(* IEC 61131-3 sources: github/IM_SYS_PRG/Code/顶出系统/托模, 2 files *)

(* ---- FB_Eject.st ---- *)
(*
  FB_Eject 功能块
  功能：
  1. 负责托模进、托模保持、托模退及其调试动作的执行状态机。
  2. 按托模参数输出压力、速度、位置命令，并返回托模进退完成状态。

  说明：
  1. 正常模式使用 1=托模进、2=托模退；调试模式使用 6/7。
  2. 组合托模模式由 `FB_EjectMode` 复用本块完成具体动作。
*)
FUNCTION_BLOCK FB_Eject
VAR_IN_OUT
    stEjectAxis: ST_AxisRefHyd;       // 托模共享轴结构
END_VAR
VAR_INPUT
    bStart: BOOL;                     // TRUE=启动托模动作
    bStop: BOOL;                      // TRUE=正常停止
    bEStop: BOOL;                     // TRUE=急停
    bReset: BOOL;                     // TRUE=复位状态机与输出
    bManualMode: BOOL;                // TRUE=手动点动托模
    uiEjectMode: UINT;                // 1=托模进 2=托模退 6=托模进调试 7=托模退调试
    stEjectPara: ST_EjectPara;        // 托模工艺参数
    bEjectInStop: BOOL;               // 托模进停止信号
    bEjectOutStop: BOOL;              // 托模退停止信号
    udiEjectElecRulerVal: UDINT;      // 位置反馈
END_VAR
VAR_OUTPUT
    bBusy: BOOL;                      // TRUE=当前动作尚未结束
    bDone: BOOL;                      // TRUE=当前动作完成
    bAlarm: BOOL;                     // TRUE=当前动作报警
    dwAlarmID: DWORD;                 // 模块报警码
    uiActHint: UINT;                  // 当前动作提示码
    uiActTime: UINT;                  // 当前动作持续时间，单位 s
    bEjectIned: BOOL;                 // TRUE=托模进完成
    bEjectOuted: BOOL;                // TRUE=托模退完成
    uiPresCmd: UINT;                  // 压力命令输出
    uiSpdCmd: UINT;                   // 速度命令输出
    udiPosCmd: UDINT;                 // 位置命令输出
END_VAR
VAR
    eState: E_EjectState := eState_Idle;
    uiStageIndex: UINT := 0;
    tPulse: TON;
    udiElapsedMs: UDINT := 0;
    bManualActive: BOOL := FALSE;
    bInRequest: BOOL := FALSE;
    bOutRequest: BOOL := FALSE;
    stSegCmd: ST_EjectSeg;
END_VAR

bManualActive := bManualMode OR (uiEjectMode = 6) OR (uiEjectMode = 7);
bInRequest := (uiEjectMode = 1) OR (uiEjectMode = 6);
bOutRequest := (uiEjectMode = 2) OR (uiEjectMode = 7);

IF bReset THEN
    eState := eState_Idle;
    bBusy := FALSE;
    bDone := FALSE;
    bAlarm := FALSE;
    dwAlarmID := 0;
    uiActHint := 0;
    uiActTime := 0;
    bEjectIned := FALSE;
    bEjectOuted := FALSE;
    uiPresCmd := 0;
    uiSpdCmd := 0;
    udiPosCmd := 0;
    uiStageIndex := 0;
    udiElapsedMs := 0;
    tPulse(IN := FALSE, PT := T#100MS);
ELSIF bEStop THEN
    eState := eState_Error;
    bAlarm := TRUE;
    dwAlarmID := dwAlarmID OR DWORD#16#0010;
    uiActHint := 1;
    uiPresCmd := 0;
    uiSpdCmd := 0;
    udiPosCmd := 0;
    tPulse(IN := FALSE, PT := T#100MS);
ELSIF bStop THEN
    eState := eState_Idle;
    bBusy := FALSE;
    uiPresCmd := 0;
    uiSpdCmd := 0;
    udiPosCmd := 0;
    uiActHint := 0;
    udiElapsedMs := 0;
    tPulse(IN := FALSE, PT := T#100MS);
ELSE
    CASE eState OF
        eState_Idle:
            bBusy := FALSE;
            bDone := FALSE;
            uiActHint := 0;
            uiActTime := 0;
            bEjectIned := FALSE;
            bEjectOuted := FALSE;
            uiPresCmd := 0;
            uiSpdCmd := 0;
            udiPosCmd := 0;
            uiStageIndex := 0;
            udiElapsedMs := 0;
            tPulse(IN := FALSE, PT := T#100MS);
            IF bStart THEN
                bAlarm := FALSE;
                dwAlarmID := 0;
                uiStageIndex := 1;
                IF bInRequest THEN
                    eState := eState_EjectIning;
                ELSIF bOutRequest THEN
                    eState := eState_EjectOuting;
                ELSE
                    bAlarm := TRUE;
                    dwAlarmID := DWORD#16#0001;
                    eState := eState_Error;
                END_IF;
            END_IF;

        eState_EjectIning:
            bBusy := TRUE;
            tPulse(IN := TRUE, PT := T#100MS);
            IF tPulse.Q THEN
                udiElapsedMs := udiElapsedMs + 100;
                tPulse(IN := FALSE, PT := T#100MS);
            END_IF;
            uiActTime := TO_UINT(udiElapsedMs / 1000);

            IF bManualActive THEN
                stSegCmd := stEjectPara.stEjectInDbgSeg;
                IF (stSegCmd.uiPres = 0) AND (stSegCmd.uiSpd = 0) AND (stSegCmd.udiPos = 0) THEN
                    stSegCmd := stEjectPara.aEjectInSeg[1];
                END_IF;
                uiActHint := 28;
                uiPresCmd := stSegCmd.uiPres;
                uiSpdCmd := stSegCmd.uiSpd;
                udiPosCmd := stSegCmd.udiPos;
                IF NOT bStart THEN
                    eState := eState_Idle;
                END_IF;
            ELSE
                IF uiStageIndex > stEjectPara.uiEjectInSegCnt THEN
                    IF stEjectPara.stEjectKeepSeg.uiTime > 0 THEN
                        eState := eState_EjectKeeping;
                    ELSE
                        eState := eState_EjectIned;
                    END_IF;
                    udiElapsedMs := 0;
                    tPulse(IN := FALSE, PT := T#100MS);
                ELSE
                    stSegCmd := stEjectPara.aEjectInSeg[uiStageIndex];
                    uiActHint := 89 + uiStageIndex; // 90-92
                    uiPresCmd := stSegCmd.uiPres;
                    uiSpdCmd := stSegCmd.uiSpd;
                    udiPosCmd := stSegCmd.udiPos;

                    IF (stEjectPara.uiEjectInMode = 2) AND (udiEjectElecRulerVal >= stSegCmd.udiPos) THEN
                        uiStageIndex := uiStageIndex + 1;
                        udiElapsedMs := 0;
                        tPulse(IN := FALSE, PT := T#100MS);
                    ELSIF ((stEjectPara.uiEjectInMode = 0) AND (stSegCmd.uiTime > 0) AND (udiElapsedMs >= TO_UDINT(stSegCmd.uiTime))) OR ((stEjectPara.uiEjectInMode = 1) AND bEjectInStop) THEN
                        uiStageIndex := uiStageIndex + 1;
                        udiElapsedMs := 0;
                        tPulse(IN := FALSE, PT := T#100MS);
                    END_IF;

                    IF (stEjectPara.uiEjectInLimitTime > 0) AND (udiElapsedMs >= TO_UDINT(stEjectPara.uiEjectInLimitTime)) THEN
                        dwAlarmID := dwAlarmID OR DWORD#16#0001;
                        eState := eState_Error;
                    END_IF;
                END_IF;
            END_IF;

        eState_EjectIned:
            bBusy := FALSE;
            bDone := TRUE;
            bEjectIned := TRUE;
            uiActHint := 30;
            uiPresCmd := 0;
            uiSpdCmd := 0;
            udiPosCmd := 0;

        eState_EjectKeeping:
            bBusy := TRUE;
            uiActHint := 29;
            uiPresCmd := stEjectPara.stEjectKeepSeg.uiPres;
            uiSpdCmd := stEjectPara.stEjectKeepSeg.uiSpd;
            udiPosCmd := stEjectPara.stEjectKeepSeg.udiPos;
            tPulse(IN := TRUE, PT := T#100MS);
            IF tPulse.Q THEN
                udiElapsedMs := udiElapsedMs + 100;
                tPulse(IN := FALSE, PT := T#100MS);
            END_IF;
            uiActTime := TO_UINT(udiElapsedMs / 1000);
            IF (stEjectPara.stEjectKeepSeg.uiTime = 0) OR (udiElapsedMs >= TO_UDINT(stEjectPara.stEjectKeepSeg.uiTime)) THEN
                eState := eState_EjectKept;
                tPulse(IN := FALSE, PT := T#100MS);
            END_IF;

        eState_EjectKept:
            bBusy := FALSE;
            bDone := TRUE;
            bEjectIned := TRUE;
            uiActHint := 29;
            uiPresCmd := 0;
            uiSpdCmd := 0;
            udiPosCmd := 0;

        eState_EjectOuting:
            bBusy := TRUE;
            tPulse(IN := TRUE, PT := T#100MS);
            IF tPulse.Q THEN
                udiElapsedMs := udiElapsedMs + 100;
                tPulse(IN := FALSE, PT := T#100MS);
            END_IF;
            uiActTime := TO_UINT(udiElapsedMs / 1000);

            IF bManualActive THEN
                stSegCmd := stEjectPara.stEjectOutDbgSeg;
                IF (stSegCmd.uiPres = 0) AND (stSegCmd.uiSpd = 0) AND (stSegCmd.udiPos = 0) THEN
                    stSegCmd := stEjectPara.aEjectOutSeg[1];
                END_IF;
                uiActHint := 31;
                uiPresCmd := stSegCmd.uiPres;
                uiSpdCmd := stSegCmd.uiSpd;
                udiPosCmd := stSegCmd.udiPos;
                IF NOT bStart THEN
                    eState := eState_Idle;
                END_IF;
            ELSE
                IF uiStageIndex > stEjectPara.uiEjectOutSegCnt THEN
                    eState := eState_EjectOuted;
                ELSE
                    stSegCmd := stEjectPara.aEjectOutSeg[uiStageIndex];
                    uiActHint := 91 + uiStageIndex; // 92-94
                    uiPresCmd := stSegCmd.uiPres;
                    uiSpdCmd := stSegCmd.uiSpd;
                    udiPosCmd := stSegCmd.udiPos;

                    IF (stEjectPara.uiEjectOutMode = 2) AND (udiEjectElecRulerVal >= stSegCmd.udiPos) THEN
                        uiStageIndex := uiStageIndex + 1;
                        udiElapsedMs := 0;
                        tPulse(IN := FALSE, PT := T#100MS);
                    ELSIF ((stEjectPara.uiEjectOutMode = 0) AND (stSegCmd.uiTime > 0) AND (udiElapsedMs >= TO_UDINT(stSegCmd.uiTime))) OR ((stEjectPara.uiEjectOutMode = 1) AND bEjectOutStop) THEN
                        uiStageIndex := uiStageIndex + 1;
                        udiElapsedMs := 0;
                        tPulse(IN := FALSE, PT := T#100MS);
                    END_IF;

                    IF (stEjectPara.uiEjectOutLimitTime > 0) AND (udiElapsedMs >= TO_UDINT(stEjectPara.uiEjectOutLimitTime)) THEN
                        dwAlarmID := dwAlarmID OR DWORD#16#0002;
                        eState := eState_Error;
                    END_IF;
                END_IF;
            END_IF;

        eState_EjectOuted:
            bBusy := FALSE;
            bDone := TRUE;
            bEjectOuted := TRUE;
            uiActHint := 32;
            uiPresCmd := 0;
            uiSpdCmd := 0;
            udiPosCmd := 0;

        eState_Error:
            bBusy := FALSE;
            bAlarm := TRUE;
            uiActHint := 1;
            uiPresCmd := 0;
            uiSpdCmd := 0;
            udiPosCmd := 0;
            tPulse(IN := FALSE, PT := T#100MS);

    ELSE
        eState := eState_Error;
    END_CASE;
END_IF;

stEjectAxis.rSetPressure := TO_LREAL(uiPresCmd);
stEjectAxis.rSetVelocity := TO_LREAL(uiSpdCmd);
stEjectAxis.rSetPosition := TO_LREAL(udiPosCmd);
stEjectAxis.stPumpRequest.bRequest := bBusy;
stEjectAxis.stPumpRequest.rPressureSet := TO_LREAL(uiPresCmd);
stEjectAxis.stPumpRequest.rFlowSet := TO_LREAL(uiSpdCmd);
IF bBusy THEN
    stEjectAxis.eAxisState := Running;
ELSE
    stEjectAxis.eAxisState := Idle;
END_IF;
stEjectAxis.nFaultCode := TO_INT(dwAlarmID);
END_FUNCTION_BLOCK

(* ---- FB_EjectMode.st ---- *)
(*
  FB_EjectMode 功能块
  功能：
  1. 在基础 `FB_Eject` 之上组合出定次、震动、停留三种托模模式。
  2. 通过内部顺序控制，把“托模进/托模退/托模保持”拼成更高层动作。
  3. 对外仍保持与普通托模模块相似的 Busy/Done/Alarm 接口，便于主控统一调用。

  说明：
  1. 本块本身不直接生成液压命令，而是复用 `FB_Eject` 完成具体动作。
  2. `uiSeqPhase` 用来表示当前执行到“复位子块、托进、再次复位、托退”的哪一步。
  3. 只有在手动组合模式被上层明确选择时，才应该让本块接管托模轴输出。
*)
FUNCTION_BLOCK FB_EjectMode
VAR_IN_OUT
    stEjectAxis: ST_AxisRefHyd;
END_VAR
VAR_INPUT
    bStart: BOOL;
    bStop: BOOL;
    bEStop: BOOL;
    bReset: BOOL;
    uiEjectMode: UINT;            // 1=定次 2=震动 3=停留
    uiEjectTimes: UINT;           // 定次/震动次数；震动模式下 0 表示持续循环
    stEjectPara: ST_EjectPara;
    bEjectInStop: BOOL;
    bEjectOutStop: BOOL;
    udiEjectElecRulerVal: UDINT;
END_VAR
VAR_OUTPUT
    bBusy: BOOL;
    bDone: BOOL;
    bAlarm: BOOL;
    dwAlarmID: DWORD;
    uiActHint: UINT;
    uiActTime: UINT;
    bEjectIned: BOOL;
    bEjectOuted: BOOL;
    uiPresCmd: UINT;
    uiSpdCmd: UINT;
    udiPosCmd: UDINT;
END_VAR
VAR
    eState: E_EjectModeState := eState_Idle;
    fbEject: FB_Eject;

    (* 发给内部 `FB_Eject` 的命令。 *)
    bCmdStart: BOOL := FALSE;
    bCmdReset: BOOL := FALSE;
    uiCmdMode: UINT := 0;

    (* 顺序控制变量。 *)
    uiExecCount: UINT := 0;
    uiSeqPhase: UINT := 0;

    (* 内部 `FB_Eject` 状态缓存。 *)
    bSubBusy: BOOL := FALSE;
    bSubDone: BOOL := FALSE;
    bSubAlarm: BOOL := FALSE;
    dwSubAlarmID: DWORD := 0;
    uiSubActHint: UINT := 0;
    uiSubActTime: UINT := 0;
    bSubEjectIned: BOOL := FALSE;
    bSubEjectOuted: BOOL := FALSE;
    uiSubPresCmd: UINT := 0;
    uiSubSpdCmd: UINT := 0;
    udiSubPosCmd: UDINT := 0;
END_VAR

(* 每个扫描周期先清空对子块的控制命令。 *)
bCmdStart := FALSE;
bCmdReset := FALSE;
uiCmdMode := 0;

IF bReset THEN
    eState := eState_Idle;
    bBusy := FALSE;
    bDone := FALSE;
    bAlarm := FALSE;
    dwAlarmID := DWORD#0;
    uiActHint := 0;
    uiActTime := 0;
    uiExecCount := 0;
    uiSeqPhase := 0;
    bCmdReset := TRUE;

ELSIF bEStop THEN
    eState := eState_Error;
    bBusy := FALSE;
    bDone := FALSE;
    bAlarm := TRUE;
    dwAlarmID := DWORD#16#0010;
    uiActHint := 1;
    uiActTime := 0;
    uiExecCount := 0;
    uiSeqPhase := 0;
    bCmdReset := TRUE;

ELSIF bStop THEN
    eState := eState_Idle;
    bBusy := FALSE;
    bDone := FALSE;
    bAlarm := FALSE;
    dwAlarmID := DWORD#0;
    uiActHint := 0;
    uiActTime := 0;
    uiExecCount := 0;
    uiSeqPhase := 0;
    bCmdReset := TRUE;

ELSE
    CASE eState OF
        eState_Idle:
            bBusy := FALSE;
            uiActHint := 0;
            uiActTime := 0;

            IF bStart THEN
                bDone := FALSE;
                bAlarm := FALSE;
                dwAlarmID := DWORD#0;
                uiExecCount := 0;
                uiSeqPhase := 0;

                CASE uiEjectMode OF
                    1: eState := eState_EjectCount;
                    2: eState := eState_EjectVibra;
                    3: eState := eState_EjectHold;
                ELSE
                    bAlarm := TRUE;
                    dwAlarmID := DWORD#16#0001;
                    eState := eState_Error;
                END_CASE;
            END_IF;

        eState_EjectCount:
            bBusy := TRUE;

            IF bSubAlarm THEN
                dwAlarmID := dwSubAlarmID;
                eState := eState_Error;
            ELSE
                CASE uiSeqPhase OF
                    0:
                        (* 子块切换动作前先复位，避免沿用上一个动作的完成态。 *)
                        bCmdReset := TRUE;
                        uiSeqPhase := 1;

                    1:
                        (* 托模进。 *)
                        uiCmdMode := 1;
                        bCmdStart := TRUE;
                        IF bSubDone THEN
                            uiSeqPhase := 2;
                        END_IF;

                    2:
                        (* 进入托模退前再复位一次子块。 *)
                        bCmdReset := TRUE;
                        uiSeqPhase := 3;

                    3:
                        (* 托模退。 *)
                        uiCmdMode := 2;
                        bCmdStart := TRUE;
                        IF bSubDone THEN
                            uiExecCount := uiExecCount + 1;
                            IF uiExecCount >= SEL(uiEjectTimes = 0, uiEjectTimes, 1) THEN
                                bBusy := FALSE;
                                bDone := TRUE;
                                eState := eState_Idle;
                            ELSE
                                uiSeqPhase := 0;
                            END_IF;
                        END_IF;

                ELSE
                    uiSeqPhase := 0;
                END_CASE;
            END_IF;

        eState_EjectVibra:
            bBusy := TRUE;

            IF bSubAlarm THEN
                dwAlarmID := dwSubAlarmID;
                eState := eState_Error;
            ELSE
                CASE uiSeqPhase OF
                    0:
                        bCmdReset := TRUE;
                        uiSeqPhase := 1;

                    1:
                        uiCmdMode := 1;
                        bCmdStart := TRUE;
                        IF bSubDone THEN
                            uiSeqPhase := 2;
                        END_IF;

                    2:
                        bCmdReset := TRUE;
                        uiSeqPhase := 3;

                    3:
                        uiCmdMode := 2;
                        bCmdStart := TRUE;
                        IF bSubDone THEN
                            uiExecCount := uiExecCount + 1;
                            IF (uiEjectTimes > 0) AND (uiExecCount >= uiEjectTimes) THEN
                                bBusy := FALSE;
                                bDone := TRUE;
                                eState := eState_Idle;
                            ELSE
                                uiSeqPhase := 0;
                            END_IF;
                        END_IF;

                ELSE
                    uiSeqPhase := 0;
                END_CASE;
            END_IF;

        eState_EjectHold:
            bBusy := TRUE;

            IF bSubAlarm THEN
                dwAlarmID := dwSubAlarmID;
                eState := eState_Error;
            ELSE
                CASE uiSeqPhase OF
                    0:
                        bCmdReset := TRUE;
                        uiSeqPhase := 1;

                    1:
                        uiCmdMode := 1;
                        bCmdStart := TRUE;
                        IF bSubDone THEN
                            bBusy := FALSE;
                            bDone := TRUE;
                            eState := eState_Idle;
                        END_IF;

                ELSE
                    uiSeqPhase := 0;
                END_CASE;
            END_IF;

        eState_Error:
            bBusy := FALSE;
            bDone := FALSE;
            bAlarm := TRUE;
            uiActHint := 1;
            IF dwAlarmID = DWORD#0 THEN
                dwAlarmID := SEL(dwSubAlarmID = DWORD#0, dwSubAlarmID, DWORD#16#0001);
            END_IF;
            bCmdReset := TRUE;

    ELSE
        dwAlarmID := DWORD#16#7FFF;
        eState := eState_Error;
    END_CASE;
END_IF;

(* 最后再调用内部子块，这样本扫描周期内刚决策出来的命令能立即送到子块。 *)
fbEject(
    stEjectAxis := stEjectAxis,
    bStart := bCmdStart,
    bStop := FALSE,
    bEStop := FALSE,
    bReset := bCmdReset,
    bManualMode := FALSE,
    uiEjectMode := uiCmdMode,
    stEjectPara := stEjectPara,
    bEjectInStop := bEjectInStop,
    bEjectOutStop := bEjectOutStop,
    udiEjectElecRulerVal := udiEjectElecRulerVal,
    bBusy => bSubBusy,
    bDone => bSubDone,
    bAlarm => bSubAlarm,
    dwAlarmID => dwSubAlarmID,
    uiActHint => uiSubActHint,
    uiActTime => uiSubActTime,
    bEjectIned => bSubEjectIned,
    bEjectOuted => bSubEjectOuted,
    uiPresCmd => uiSubPresCmd,
    uiSpdCmd => uiSubSpdCmd,
    udiPosCmd => udiSubPosCmd
);

(* 对外透传内部托模块的实际动作输出，便于主控统一读取。 *)
bEjectIned := bSubEjectIned;
bEjectOuted := bSubEjectOuted;
uiPresCmd := uiSubPresCmd;
uiSpdCmd := uiSubSpdCmd;
udiPosCmd := udiSubPosCmd;

IF (NOT bAlarm) AND (uiSubActHint <> 0) THEN
    uiActHint := uiSubActHint;
END_IF;
uiActTime := uiSubActTime;
END_FUNCTION_BLOCK
